PROGRAM MAIN
VAR
	
	test : BOOL;
	test2 : BOOL;
END_VAR

//CHECK

END_PROGRAM

(* stored: Version 1.1.0.1, ProductVersion 3.1.4024.9
   POU MAIN: Id {d2bfc508-792e-4c16-984e-6b9cb488ac84}, SpecialFunc None *)
